(*NOTES TO SETUP VIRTUAL AXIS:
For the virtual axis setup, the encoders need their type changed from "simulation encoder" to "Encoder (Universal)".
In addition the scale factor needs to be changed to a numerator of 1 and denominator of fEncoderScaling which is 10,000 by default)
Care needs to be taken with scaling and setup of both real and virtual axes to ensure velocities are not too fast and axes have time to settle before they submit a "complete move"
Link the virtual encoder inputs to the Gap and Centre position calculations nGapSizePosition and nGapCentrePosition
Encoder needs to be set as ABSOLUTE
Encoder Mask has to be set to 0xFFFFFFFF otherwise UDINT will overflow
NOTES TO FB_SlitPair:
The instance of the function block should be called before the call of FB_Axis, so that it gets bExecute before FB_Axis
*)
FUNCTION_BLOCK FB_SlitPair
VAR_IN_OUT
    stBladeNegative: ST_AxisStruct; //Axis data of the negative blade
    stBladePositive: ST_AxisStruct; //Axis data of the positive blade
    stGapSize: ST_AxisStruct; //Axis data of the gap size
    stGapCentre: ST_AxisStruct; //Axis data of the gap centre
END_VAR
VAR_INPUT
    iGapSize: UINT; //Axis ID for the size of gap between slit blades
    iGapCentre: UINT; //Axis ID for the centre position of the gap formed by slit blades
    fEncoderScaling: LREAL := 10000.0; //default scaling denominator of 10000
    bAutoHome: BOOL := FALSE; //Blades homing is automatically done if they are not homed
    bAnticollisionEnable: BOOL := TRUE; //Blades anticollision option, only for when blades are moved independently
    fAnticollisionMargin: LREAL := 5.0; //Margin between the the blades for anticollision
END_VAR
VAR_OUTPUT
    bEnabled: BOOL := FALSE; //Enabled status of function
    bError: BOOL; //Error status of function
    bHoming: BOOL := FALSE; //TRUE if function is homing axes
END_VAR
VAR
    //Internal state machines
    eSlitPairState: E_SlitPairStates := E_SlitPairStates.eStartup; //Sequence steps for operating the slits
    eParameterCheck: E_AxisParamCheckState := E_AxisParamCheckState.eInit; //Sequence steps for checking params of virtual axes
    eSoftLimitsUpdate: E_SlitSoftLimits := E_SlitSoftLimits.eStart; //Sequence steps for update of soft limits for virtual axes

    //Internal statuses for logic
    bEnable: BOOL; //Enable/disable the slit set
    bReset: BOOL; //Reset the slit set
    bResetting: BOOL := FALSE; //TRUE if axis going through a reset
    bAxesEnabled: BOOL := FALSE; //TRUE if all axes enabled
    bBladesHomed: BOOL := FALSE; //TRUE if blade axes are calibrated
    bGapHomed: BOOL := FALSE; //TRUE if virtual axes are calibrated
    bBladesCoupled: BOOL := FALSE; //TRUE if both blade axes are coupled
    bBladesUncoupled: BOOL := FALSE; //TRUE if both blade axes are uncoupled
    bAxisErrorsPresent: BOOL := FALSE; //TRUE if error present on any real or virtual axis
    bUpdateSoftLimits: BOOL := FALSE; //TRUE if update of soft limits are being executed
    bHomingRequested: BOOL := FALSE; //TRUE if homing is requested for all axis
    bInvalidParamFound: BOOL := FALSE; //TRUE if startup finds atleast one invalid parameter
    fGapSizePosition: LREAL; //Virtual axis gap size calculated position
    nGapSizePosition AT %Q*: UDINT := 0; //Virtual axis gap size encoder position/counter
    fGapCentrePosition: LREAL; //Virtual axis gap centre calculated position
    nGapCentrePosition AT %Q*: UDINT := 0; //Virtual axis gap centre encoder position/counter
    nAutoErrorResetCounter: UINT := 0; //Error automatic reset counter
    iParamCheck: USINT := 1; //Index of current parameter to be validated
    rtrigSlitOperational: R_TRIG;
    rtrigVirtualAxisEnable: R_TRIG;
    rtrigVirtualAxisDisable: R_TRIG;
    rtrigVirtualAxisNotMoving: R_TRIG;
    fbResetCalibrationPositiveBlade: MC_Home;
    fbResetCalibrationNegativeBlade: MC_Home;
    fbResetCalibrationGapSize: MC_Home;
    fbResetCalibrationGapCentre: MC_Home;
END_VAR
VAR CONSTANT
    cSoftLimitDelta: LREAL := 0.05; //Delta between the softlimits of physical and virtual axes
    cMaxParams: USINT := 6;
    cParameters: ARRAY [1..cMaxParams] OF ST_AxisParamSpec := [ //Parameters required to be validated
        (eParam := E_AxisParameters.AxisEncoderScalingNumerator, fValue := 1.0),
        (eParam := E_AxisParameters.AxisEncoderScalingDenominator, fValue := 10000.0),
        (eParam := E_AxisParameters.AxisEncoderMask, fValue := 4294967295.0), //0xFFFFFFF = 4294967295.0
        (eParam := E_AxisParameters.AxisEncoderReferenceSystem, fValue := 1.0), //0.0 = INCREMENTAL, 1.0 = ABSOLUTE
        (eParam := E_AxisParameters.EnableLimitBackward, fValue := 1.0), //0.0 = FALSE, 1.0 = TRUE
        (eParam := E_AxisParameters.EnableLimitForward, fValue := 1.0)]; //0.0 = FALSE, 1.0 = TRUE
END_VAR

//Configure homing routine of virtual axes
stGapSize.stConfig.eHomeSeq := E_HomingRoutines.eHomeDirect;
stGapCentre.stConfig.eHomeSeq := E_HomingRoutines.eHomeDirect;

//Run actions for slit set
actErrorHandling(); //Error handling subroutine
actGapLimits(); //Set virtual axis limits to TRUE
actVirtualAxisPositions(); //Virtual axis encoder position subroutine
actUpdateStatus(); //Update statuses
actEnableAxes(); //Enable the axes
actClearCalibration(); //Clear calibration flag for all axes
mAnticollision(
    stBladeNegative := stBladeNegative,
    stBladePositive := stBladePositive); //Handle blades anticollision

CASE eSlitPairState OF
    E_SlitPairStates.eStartup:
        checkStartupParams(stGapSize, stGapCentre);
        IF eParameterCheck = E_AxisParamCheckState.eFinish THEN
            eSlitPairState := E_SlitPairStates.eInit;
        END_IF

    E_SlitPairStates.eInit:
        bEnabled := FALSE;
        IF bAxesEnabled AND bEnable THEN
            eSlitPairState := E_SlitPairStates.eInitClearGearing;
        END_IF

    E_SlitPairStates.eInitClearGearing:
        actClearSlitGearing();
        eSlitPairState := E_SlitPairStates.eInitGearOutCheck;

    E_SlitPairStates.eInitGearOutCheck: //Check gearout completion
        IF bBladesUncoupled THEN
            eSlitPairState := E_SlitPairStates.eCheckHomeStatus;
        END_IF

    E_SlitPairStates.eCheckHomeStatus: //If blades are already homed, skip to virtual homing, otherwise wait for manual/auto homing signal
        IF bBladesHomed THEN
            eSlitPairState := E_SlitPairStates.eHomeGap; //Skip to functioning
        ELSIF bAutoHome
            OR bHomingRequested
            OR (stGapSize.stControl.eCommand = E_MotionFunctions.eHome AND stGapSize.stControl.bExecute)
            OR (stGapCentre.stControl.eCommand = E_MotionFunctions.eHome AND stGapCentre.stControl.bExecute)
        THEN
            bHomingRequested := FALSE; //If homing fails do not automatically start homing again
            eSlitPairState := E_SlitPairStates.eHomeBlades;
        END_IF

    E_SlitPairStates.eHomeBlades: //Initiate homing of blade axes. Homing routine must be pre-configured by user
        stBladeNegative.stControl.eCommand := E_MotionFunctions.eHome;
        stBladePositive.stControl.eCommand := E_MotionFunctions.eHome;
        stBladeNegative.stControl.bExecute := TRUE;
        stBladePositive.stControl.bExecute := TRUE;
        bHoming := TRUE;
        eSlitPairState := E_SlitPairStates.eCheckBladeHomeComplete;

    E_SlitPairStates.eCheckBladeHomeComplete: //Wait for completion of blade homing routines or stop/halt command
        IF bBladesHomed AND NOT stBladeNegative.stStatus.bBusy AND NOT stBladePositive.stStatus.bBusy THEN
            eSlitPairState := E_SlitPairStates.eHomeGap;
            bHoming := FALSE;
        ELSIF stGapSize.stControl.bStop OR stGapCentre.stControl.bStop THEN
            stBladeNegative.stControl.bStop := TRUE;
            stBladePositive.stControl.bStop := TRUE;
            eSlitPairState := E_SlitPairStates.eCheckHomeStatus;
        ELSIF stGapSize.stControl.bHalt OR stGapCentre.stControl.bHalt THEN
            stBladeNegative.stControl.bHalt := TRUE;
            stBladePositive.stControl.bHalt := TRUE;
            eSlitPairState := E_SlitPairStates.eCheckHomeStatus;
        ELSIF (stBladeNegative.stStatus.nErrorID > 0) OR (stBladePositive.stStatus.nErrorID > 0) THEN
            eSlitPairState := E_SlitPairStates.eError;
        END_IF

    E_SlitPairStates.eHomeGap: //"Home" the virtual axes
        stGapSize.stConfig.eHomeSeq := E_HomingRoutines.eHomeDirect;
        stGapCentre.stConfig.eHomeSeq := E_HomingRoutines.eHomeDirect;
        stGapSize.stConfig.fHomePosition := fGapSizePosition;
        stGapCentre.stConfig.fHomePosition := fGapCentrePosition;
        stGapSize.stControl.eCommand := E_MotionFunctions.eHome;
        stGapCentre.stControl.eCommand := E_MotionFunctions.eHome;
        stGapSize.stControl.bExecute := TRUE;
        stGapCentre.stControl.bExecute := TRUE;
        eSlitPairState := E_SlitPairStates.eCheckGapHomeComplete;

    E_SlitPairStates.eCheckGapHomeComplete: //Wait for virtual homing completion
        IF bGapHomed AND NOT stGapSize.stStatus.bBusy AND NOT stGapCentre.stStatus.bBusy THEN
            eSlitPairState := E_SlitPairStates.eGearInSlits;
        END_IF

    E_SlitPairStates.eGearInSlits: //Setup gearing
        actSetupSlitGearing();
        eSlitPairState := E_SlitPairStates.eCheckGearInSlitsComplete;

    E_SlitPairStates.eCheckGearInSlitsComplete: //Wait for gearing complete
        IF bBladesCoupled THEN
            eSlitPairState := E_SlitPairStates.eSlitsOperational;
        ELSIF NOT stGapSize.stStatus.bEnabled AND NOT stGapCentre.stStatus.bEnabled THEN
            eSlitPairState := E_SlitPairStates.eErrorGearOut;
        END_IF

    E_SlitPairStates.eSlitsOperational: //SLITS OPERATIONAL - Monitor for any gear outs and re-gear when no busy blades
        bEnabled := TRUE;
        checkSoftLimits(stGapSize, stGapCentre); //Soft limits are updated when axes are stopped
        IF (NOT bBladesCoupled OR NOT bEnable) AND NOT stBladeNegative.stStatus.bBusy AND NOT stBladePositive.stStatus.bBusy THEN
            eSlitPairState := E_SlitPairStates.eGearOutBlades;
        END_IF
        IF (stGapSize.stControl.eCommand = E_MotionFunctions.eHome AND stGapSize.stControl.bExecute) OR
            (stGapCentre.stControl.eCommand = E_MotionFunctions.eHome AND stGapCentre.stControl.bExecute) THEN
            eSlitPairState := E_SlitPairStates.eGearOutBlades;
            bHomingRequested := TRUE;
        END_IF

    E_SlitPairStates.eGearOutBlades: //Clear any residual gearing
        actClearSlitGearing();
        eSlitPairState := E_SlitPairStates.eCheckGearOutComplete;

    E_SlitPairStates.eCheckGearOutComplete: //Check gearing cleared
        IF bBladesUncoupled THEN
            IF bHomingRequested THEN
                eSlitPairState := E_SlitPairStates.eResetCalibration;
                bEnabled := FALSE;
            ELSE
                eSlitPairState := E_SlitPairStates.eInit;
            END_IF
        END_IF

    E_SlitPairStates.eResetCalibration:
        IF checkResetCalibrationDone() THEN
            eSlitPairState := E_SlitPairStates.eCheckHomeStatus;
        ELSIF checkResetCalibrationFailed() THEN
            eSlitPairState := E_SlitPairStates.eError;
        END_IF

    E_SlitPairStates.eError: //ERROR STATE
        nAutoErrorResetCounter := 0;
        bError := TRUE;
        bEnabled := FALSE;
        IF bReset THEN
            bResetting := TRUE;
            eSlitPairState := E_SlitPairStates.eErrorGearOut;
        END_IF

    E_SlitPairStates.eErrorGearOut: //Try to clear issues
        actClearSlitGearing();
        eSlitPairState := E_SlitPairStates.eErrorGearOutCheck;

    E_SlitPairStates.eErrorGearOutCheck:
        IF bBladesUncoupled THEN
            eSlitPairState := E_SlitPairStates.eErrorResetAxes;
        END_IF

    E_SlitPairStates.eErrorResetAxes: //RESET ALL AXES
        stBladeNegative.stControl.bReset := TRUE;
        stBladePositive.stControl.bReset := TRUE;
        stGapSize.stControl.bReset := TRUE;
        stGapCentre.stControl.bReset := TRUE;
        nAutoErrorResetCounter := nAutoErrorResetCounter + 1;
        eSlitPairState := E_SlitPairStates.eErrorResetCheck;

    E_SlitPairStates.eErrorResetCheck:
        IF bAxisErrorsPresent THEN
            //If the errors persists after 10 auto reset, then manual intervention is required
            IF nAutoErrorResetCounter <= 10 THEN
                eSlitPairState := E_SlitPairStates.eErrorResetAxes;
            END_IF
        ELSE
            eSlitPairState := E_SlitPairStates.eInit;
            nAutoErrorResetCounter := 0;
            bError := FALSE;
            bResetting := FALSE;
        END_IF
END_CASE

bReset := FALSE;

ACTION actClearCalibration:
fbResetCalibrationPositiveBlade(
    Axis := stBladePositive.Axis,
    Execute := eSlitPairState = E_SlitPairStates.eResetCalibration,
    HomingMode := MC_HomingMode.MC_ResetCalibration);

fbResetCalibrationNegativeBlade(
    Axis := stBladeNegative.Axis,
    Execute := eSlitPairState = E_SlitPairStates.eResetCalibration,
    HomingMode := MC_HomingMode.MC_ResetCalibration);

fbResetCalibrationGapSize(
    Axis := stGapSize.Axis,
    Execute := eSlitPairState = E_SlitPairStates.eResetCalibration,
    HomingMode := MC_HomingMode.MC_ResetCalibration);

fbResetCalibrationGapCentre(
    Axis := stGapCentre.Axis,
    Execute := eSlitPairState = E_SlitPairStates.eResetCalibration,
    HomingMode := MC_HomingMode.MC_ResetCalibration);
END_ACTION

ACTION actClearSlitGearing:
//Action to send gearOut command to blade axes
stBladeNegative.stControl.eCommand := E_MotionFunctions.eGearOut;
stBladePositive.stControl.eCommand := E_MotionFunctions.eGearOut;
stBladeNegative.stControl.bExecute := TRUE;
stBladePositive.stControl.bExecute := TRUE;
END_ACTION

ACTION actEnableAxes:
//Enable all axes when one of the virtual axes is enabled
rtrigVirtualAxisEnable(CLK := stGapSize.stControl.bEnable OR stGapCentre.stControl.bEnable);

IF rtrigVirtualAxisEnable.Q THEN
    stBladePositive.stControl.bEnable := TRUE;
    stBladeNegative.stControl.bEnable := TRUE;
    stGapSize.stControl.bEnable := TRUE;
    stGapCentre.stControl.bEnable := TRUE;
    bEnable := TRUE;
END_IF

//Disable blade axes when both the virtuals are disabled
rtrigVirtualAxisDisable(CLK := NOT stGapSize.stControl.bEnable OR NOT stGapCentre.stControl.bEnable);

IF rtrigVirtualAxisDisable.Q THEN
    stBladePositive.stControl.bEnable := FALSE;
    stBladeNegative.stControl.bEnable := FALSE;
    stGapSize.stControl.bEnable := FALSE;
    stGapCentre.stControl.bEnable := FALSE;
END_IF

//Set Enable flag when all axes are enabled
bEnable := stBladePositive.stStatus.bEnabled AND stBladeNegative.stStatus.bEnabled
    AND stGapSize.stStatus.bEnabled AND stGapCentre.stStatus.bEnabled;
END_ACTION

ACTION actErrorHandling:
//Error handling for slit functionality
IF bResetting THEN //ignore setting in error state if FB going through a reset
    RETURN;
END_IF

//RESET - Use the reset from the virtual axes in order to reset the slits
bReset := stGapCentre.stControl.bReset OR stGapSize.stControl.bReset;

IF NOT bError AND bAxisErrorsPresent AND (stGapCentre.stStatus.bEnabled OR stGapSize.stStatus.bEnabled) THEN
    actStopAxes();
    eSlitPairState := E_SlitPairStates.eError;
END_IF

//Report error to virtual axes
IF eSlitPairState = E_SlitPairStates.eError THEN
    stGapCentre.stStatus.bError := TRUE;
    stGapSize.stStatus.bError := TRUE;
END_IF

IF bEnabled AND NOT bBladesHomed THEN
    eSlitPairState := E_SlitPairStates.eError;
END_IF
END_ACTION

ACTION actGapLimits:
//Set Virtual axes inputs to TRUE to enable movement
stGapSize.stInputs.bLimitBwd := stBladeNegative.stInputs.bLimitFwd OR stBladePositive.stInputs.bLimitBwd;
stGapSize.stInputs.bLimitFwd := stBladeNegative.stInputs.bLimitBwd OR stBladePositive.stInputs.bLimitFwd;
stGapCentre.stInputs.bLimitBwd := stBladeNegative.stInputs.bLimitFwd OR stBladePositive.stInputs.bLimitBwd;
stGapCentre.stInputs.bLimitFwd := stBladeNegative.stInputs.bLimitBwd OR stBladePositive.stInputs.bLimitFwd;
END_ACTION

ACTION actSetupSlitGearing:
//Setup multimaster gearing of negative blade
stBladeNegative.stControl.eCommand := E_MotionFunctions.eGearInMultiMaster;
stBladeNegative.stConfig.astMultiMasterAxis[1].nIndex := iGapSize;
stBladeNegative.stConfig.astMultiMasterAxis[1].fRatio := -0.5;
stBladeNegative.stConfig.astMultiMasterAxis[2].nIndex := iGapCentre;
stBladeNegative.stConfig.astMultiMasterAxis[2].fRatio := 1.0;
stBladeNegative.stConfig.astMultiMasterAxis[3].nIndex := iGapCentre;
stBladeNegative.stConfig.astMultiMasterAxis[3].fRatio := 0.0;
stBladeNegative.stConfig.astMultiMasterAxis[4].nIndex := iGapCentre;
stBladeNegative.stConfig.astMultiMasterAxis[4].fRatio := 0.0;
//Setup multimaster gearing of positive blade
stBladePositive.stControl.eCommand := E_MotionFunctions.eGearInMultiMaster;
stBladePositive.stConfig.astMultiMasterAxis[1].nIndex := iGapSize;
stBladePositive.stConfig.astMultiMasterAxis[1].fRatio := 0.5;
stBladePositive.stConfig.astMultiMasterAxis[2].nIndex := iGapCentre;
stBladePositive.stConfig.astMultiMasterAxis[2].fRatio := 1.0;
stBladePositive.stConfig.astMultiMasterAxis[3].nIndex := iGapCentre;
stBladePositive.stConfig.astMultiMasterAxis[3].fRatio := 0.0;
stBladePositive.stConfig.astMultiMasterAxis[4].nIndex := iGapCentre;
stBladePositive.stConfig.astMultiMasterAxis[4].fRatio := 0.0;
//Execute
stBladeNegative.stControl.bExecute := TRUE;
stBladePositive.stControl.bExecute := TRUE;
END_ACTION

ACTION actStopAxes:
//Stop all axes when in error (Abort movements)
stBladePositive.stControl.bStop := TRUE;
stBladeNegative.stControl.bStop := TRUE;
stGapSize.stControl.bStop := TRUE;
stGapCentre.stControl.bStop := TRUE;
END_ACTION

ACTION actUpdateSoftLimits:
//The soft limits of the virtual axes are updated everytime a movement has been accomplished.
//This is to avoid undesired errors if the user sets a target position which is not allowed

CASE eSoftLimitsUpdate OF

    E_SlitSoftLimits.eStart:
        eSoftLimitsUpdate := E_SlitSoftLimits.eWriteGapCentreFwd;

    E_SlitSoftLimits.eWriteGapCentreFwd:
        IF NOT stGapCentre.stStatus.bBusy AND NOT stGapSize.stStatus.bBusy THEN
            eSoftLimitsUpdate := E_SlitSoftLimits.eWriteGapCentreBwd;
            stGapCentre.stControl.bExecute := TRUE;
            stGapCentre.stControl.eCommand := E_MotionFunctions.eWriteParameter;
            stGapCentre.stConfig.eAxisParameters := E_AxisParameters.SWLimitForward;
            stGapCentre.stConfig.fWriteAxisParameter := stBladePositive.stConfig.fMaxSoftPosLimit
                - ABS(stGapCentre.stStatus.fActPosition - stBladePositive.stStatus.fActPosition)
                - cSoftLimitDelta;
        END_IF

    E_SlitSoftLimits.eWriteGapCentreBwd:
        IF stGapCentre.stStatus.bDone AND NOT stGapCentre.stControl.bExecute THEN
            eSoftLimitsUpdate := E_SlitSoftLimits.eWriteGapSizeFwd;
            stGapCentre.stControl.bExecute := TRUE;
            stGapCentre.stControl.eCommand := E_MotionFunctions.eWriteParameter;
            stGapCentre.stConfig.eAxisParameters := E_AxisParameters.SWLimitBackward;
            stGapCentre.stConfig.fWriteAxisParameter := stBladeNegative.stConfig.fMinSoftPosLimit
                + ABS(stGapCentre.stStatus.fActPosition - stBladeNegative.stStatus.fActPosition)
                + cSoftLimitDelta;
        END_IF

    E_SlitSoftLimits.eWriteGapSizeFwd:
        IF stGapCentre.stStatus.bDone AND NOT stGapCentre.stControl.bExecute THEN
            eSoftLimitsUpdate := E_SlitSoftLimits.eFinish;
            stGapSize.stControl.bExecute := TRUE;
            stGapSize.stControl.eCommand := E_MotionFunctions.eWriteParameter;
            stGapSize.stConfig.eAxisParameters := E_AxisParameters.SWLimitForward;
            stGapSize.stConfig.fWriteAxisParameter := 2.0 * MAX(MIN(
                ABS(stBladePositive.stConfig.fMaxSoftPosLimit - stGapCentre.stStatus.fActPosition),
                ABS(stBladeNegative.stConfig.fMinSoftPosLimit - stGapCentre.stStatus.fActPosition))
                - cSoftLimitDelta,
                0.0);
        END_IF

    E_SlitSoftLimits.eFinish:
        IF stGapSize.stStatus.bDone AND NOT stGapSize.stControl.bExecute THEN
            eSoftLimitsUpdate := E_SlitSoftLimits.eStart;
            bUpdateSoftLimits := FALSE;
        END_IF

END_CASE
END_ACTION

ACTION actUpdateStatus:
bAxesEnabled := checkAllAxesEnabled(stBladeNegative, stBladePositive, stGapSize, stGapCentre);
bBladesHomed := checkBladesHomed(stBladeNegative, stBladePositive);
bGapHomed := checkGapHomed(stGapSize, stGapCentre);
bBladesCoupled := checkBladesCoupled(stBladeNegative, stBladePositive);
bBladesUncoupled := checkBladesUncoupled(stBladeNegative, stBladePositive);
bAxisErrorsPresent := checkAnyAxisHasError(stBladeNegative, stBladePositive, stGapSize, stGapCentre);
END_ACTION

ACTION actVirtualAxisPositions:
(*Calculate virtual axes positions and convert to UDINT.
Conversion to UDINT is prohibited if it would exceed UDINT max value of 4,294,967,295.
If this is not done, it can cause overflow when connected to the encoder input and hard-crash the PLC which will only recover with a power cycle.
To preserve decimal position data of the LREAL (i.e. anything <1mm) it is necessary to scale the value before converting to UDINT.
This can be reversed with the correct scaling at the NC encoder level.
*)
fGapSizePosition := stBladePositive.stStatus.fActPosition - stBladeNegative.stStatus.fActPosition;
fGapCentrePosition := (stBladePositive.stStatus.fActPosition + stBladeNegative.stStatus.fActPosition) / 2;

IF bBladesHomed THEN
    IF ABS(fGapSizePosition) < 100000 THEN
        nGapSizePosition := LREAL_TO_UDINT(fGapSizePosition*fEncoderScaling);
    END_IF
    IF ABS(fGapCentrePosition) < 100000 THEN
        nGapCentrePosition := LREAL_TO_UDINT(fGapCentrePosition*fEncoderScaling);
    END_IF
END_IF
END_ACTION

(*Method to check if all axes (real and virtual) are enabled.
Only returns TRUE if BOTH blades are homed*)
METHOD PRIVATE checkAllAxesEnabled: BOOL
VAR_IN_OUT
    stBladeNegative: ST_AxisStruct; //Axis data of the negative blade
    stBladePositive: ST_AxisStruct; //Axis data of the positive blade
    stGapSize: ST_AxisStruct; //Axis data of the gap size
    stGapCentre: ST_AxisStruct; //Axis data of the gap centre
END_VAR
checkAllAxesEnabled := stBladeNegative.stStatus.bEnabled
    AND stBladePositive.stStatus.bEnabled
    AND stGapSize.stStatus.bEnabled
    AND stGapCentre.stStatus.bEnabled;
END_METHOD

(*Method to check if an error is present on any axis.
Returns TRUE if an error is present on any axis *)
METHOD PRIVATE checkAnyAxisHasError: BOOL
VAR_IN_OUT
    stBladeNegative: ST_AxisStruct; //Axis data of the negative blade
    stBladePositive: ST_AxisStruct; //Axis data of the positive blade
    stGapSize: ST_AxisStruct; //Axis data of the gap size
    stGapCentre: ST_AxisStruct; //Axis data of the gap centre
END_VAR
checkAnyAxisHasError := stGapSize.stStatus.bError
    OR stGapCentre.stStatus.bError
    OR stBladeNegative.stStatus.bError
    OR stBladePositive.stStatus.bError;
END_METHOD

(*Method to check if both blades are coupled to the virtual axes.
Only returns TRUE if BOTH blades are coupled *)
METHOD PRIVATE checkBladesCoupled: BOOL
VAR_IN_OUT
    stBladeNegative: ST_AxisStruct; //Axis data of the negative blade
    stBladePositive: ST_AxisStruct; //Axis data of the positive blade
END_VAR
checkBladesCoupled := stBladeNegative.stStatus.bGeared AND stBladePositive.stStatus.bGeared;
END_METHOD

(*Method to check if blade axes are homed/have the calibration flag.
Only returns TRUE if BOTH blades are homed*)
METHOD PRIVATE checkBladesHomed: BOOL
VAR_IN_OUT
    stBladeNegative: ST_AxisStruct; //Axis data of the negative blade
    stBladePositive: ST_AxisStruct; //Axis data of the positive blade
END_VAR
checkBladesHomed := stBladeNegative.stStatus.bHomed AND stBladePositive.stStatus.bHomed;
END_METHOD

(*Method to check if both blades are uncoupled from the virtual axes.
Only returns TRUE if BOTH blades are uncoupled *)
METHOD PRIVATE checkBladesUncoupled: BOOL
VAR_IN_OUT
    stBladeNegative: ST_AxisStruct; //Axis data of the negative blade
    stBladePositive: ST_AxisStruct; //Axis data of the positive blade
END_VAR
checkBladesUncoupled := NOT (stBladeNegative.stStatus.bGeared OR stBladePositive.stStatus.bGeared);
END_METHOD

(*Method to check if the virtual axes for gap size and gap centre are homed/the calibration flag is present.
Only returns TRUE if BOTH virtual axes are homed *)
METHOD PRIVATE checkGapHomed: BOOL
VAR_IN_OUT
    stGapSize: ST_AxisStruct; //Axis data of the gap size
    stGapCentre: ST_AxisStruct; //Axis data of the gap size
END_VAR
checkGapHomed := stGapSize.stStatus.bHomed AND stGapCentre.stStatus.bHomed;
END_METHOD

METHOD PRIVATE checkResetCalibrationDone : BOOL
VAR_INPUT
END_VAR
checkResetCalibrationDone := NOT fbResetCalibrationPositiveBlade.Busy
    AND NOT fbResetCalibrationNegativeBlade.Busy
    AND NOT fbResetCalibrationGapSize.Busy
    AND NOT fbResetCalibrationGapCentre.Busy
    AND NOT bBladesHomed
    AND NOT bGapHomed;
END_METHOD

METHOD PRIVATE checkResetCalibrationFailed : BOOL
VAR_INPUT
END_VAR
checkResetCalibrationFailed := fbResetCalibrationPositiveBlade.Error
    OR fbResetCalibrationNegativeBlade.Error
    OR fbResetCalibrationGapSize.Error
    OR fbResetCalibrationGapCentre.Error
    OR fbResetCalibrationPositiveBlade.CommandAborted
    OR fbResetCalibrationNegativeBlade.CommandAborted
    OR fbResetCalibrationGapSize.CommandAborted
    OR fbResetCalibrationGapCentre.CommandAborted;
END_METHOD

METHOD PRIVATE checkSoftLimits
VAR_IN_OUT
    stGapSize: ST_AxisStruct; //Axis data of the gap size
    stGapCentre: ST_AxisStruct; //Axis data of the gap centre
END_VAR
rtrigVirtualAxisNotMoving(CLK := NOT stGapCentre.stStatus.bMoving AND NOT stGapSize.stStatus.bMoving);
rtrigSlitOperational(CLK := eSlitPairState = E_SlitPairStates.eSlitsOperational);

IF rtrigVirtualAxisNotMoving.Q OR rtrigSlitOperational.Q THEN
    bUpdateSoftLimits := TRUE;
END_IF

IF bUpdateSoftLimits THEN
    actUpdateSoftLimits();
END_IF
END_METHOD

METHOD PRIVATE checkStartupParams
VAR_IN_OUT
    stGapSize: ST_AxisStruct; //Axis data of the gap size
    stGapCentre: ST_AxisStruct; //Axis data of the gap centre
END_VAR
VAR
    sWarnMsg: T_MaxString;
END_VAR
CASE eParameterCheck OF
    E_AxisParamCheckState.eInit:
        //Wait for axis initialization
        IF NOT (stGapSize.stStatus.bAxisInitialized AND stGapCentre.stStatus.bAxisInitialized) THEN
            RETURN;
        END_IF

        iParamCheck := 1;
        eParameterCheck := E_AxisParamCheckState.eSelectParam;

    E_AxisParamCheckState.eSelectParam:
        stGapSize.stConfig.eAxisParameters := cParameters[iParamCheck].eParam;
        stGapSize.stControl.eCommand := E_MotionFunctions.eReadParameter;
        stGapSize.stControl.bExecute := TRUE;

        stGapCentre.stConfig.eAxisParameters := cParameters[iParamCheck].eParam;
        stGapCentre.stControl.eCommand := E_MotionFunctions.eReadParameter;
        stGapCentre.stControl.bExecute := TRUE;

        eParameterCheck := E_AxisParamCheckState.eWaitRead;

    E_AxisParamCheckState.eWaitRead:
        //Parameter reading still in progress
        IF stGapSize.stStatus.bBusy OR stGapCentre.stStatus.bBusy THEN
            RETURN;
        END_IF

        eParameterCheck := E_AxisParamCheckState.eCheck;

    E_AxisParamCheckState.eCheck:
        IF stGapSize.stConfig.fReadAxisParameter = cParameters[iParamCheck].fValue
            AND stGapCentre.stConfig.fReadAxisParameter = cParameters[iParamCheck].fValue
        THEN
            eParameterCheck := E_AxisParamCheckState.eParamValid;
        ELSE
            eParameterCheck := E_AxisParamCheckState.eParamInvalid;
        END_IF

    E_AxisParamCheckState.eParamValid:
        eParameterCheck := E_AxisParamCheckState.eNext;

    E_AxisParamCheckState.eParamInvalid:
        //Gap Size
        IF stGapSize.stConfig.fReadAxisParameter <> cParameters[iParamCheck].fValue THEN
            sWarnMsg := CONCAT(
                STR1 := 'Slit virtual axis Gap Size (AxisId=%d) has an invalid parameter of ',
                STR2 := TO_STRING(cParameters[iParamCheck].eParam));

            ADSLOGDINT(
                msgCtrlMask := ADSLOG_MSGTYPE_WARN,
                msgFmtStr := sWarnMsg,
                dintArg := TO_DINT(iGapSize));
        END_IF
        //Gap Centre
        IF stGapCentre.stConfig.fReadAxisParameter <> cParameters[iParamCheck].fValue THEN
            sWarnMsg := CONCAT(
                STR1 := 'Slit virtual axis Gap Centre (AxisId=%d) has an invalid parameter of ',
                STR2 := TO_STRING(cParameters[iParamCheck].eParam));

            ADSLOGDINT(
                msgCtrlMask := ADSLOG_MSGTYPE_WARN,
                msgFmtStr := sWarnMsg,
                dintArg := TO_DINT(iGapCentre));
        END_IF
        bInvalidParamFound := TRUE;

        eParameterCheck := E_AxisParamCheckState.eNext;

    E_AxisParamCheckState.eNext:
        IF iParamCheck = cMaxParams THEN
            IF NOT bInvalidParamFound THEN
                ADSLOGSTR(
                    msgCtrlMask := ADSLOG_MSGTYPE_LOG,
                    msgFmtStr := 'Slit all parameters of both virtual axes are valid',
                    strArg := '');
            END_IF
            eParameterCheck := E_AxisParamCheckState.eFinish;
        ELSE
            ;
            iParamCheck := iParamCheck + 1;
            eParameterCheck := E_AxisParamCheckState.eSelectParam;
        END_IF


    E_AxisParamCheckState.eFinish:
        ;

END_CASE
END_METHOD

METHOD PRIVATE mAntiCollision
VAR_IN_OUT
    stBladeNegative: ST_AxisStruct; //Axis data of the negative blade
    stBladePositive: ST_AxisStruct; //Axis data of the positive blade
END_VAR
VAR
    fNegativeBladePosWithMargin: LREAL;
    fPositiveBladePosWithMargin: LREAL;
END_VAR
//Return early if preconditions are not met
IF NOT (bBladesHomed
    AND bBladesUncoupled
    AND bAnticollisionEnable)
THEN
    RETURN;
END_IF

//Negative Blade

fPositiveBladePosWithMargin := (stBladePositive.stStatus.fActPosition - fAnticollisionMargin);

//If executing absolute / relative movement commands also check target position
IF stBladeNegative.stControl.bExecute THEN
    CASE stBladeNegative.stControl.eCommand OF

        E_MotionFunctions.eMoveAbsolute:
            stBladeNegative.stControl.bInterlockFwd S= stBladeNegative.stControl.fPosition
                >= fPositiveBladePosWithMargin;

        E_MotionFunctions.eMoveRelative:
            stBladeNegative.stControl.bInterlockFwd S= (stBladeNegative.stControl.fPosition
                + stBladeNegative.stStatus.fActPosition)
                >= fPositiveBladePosWithMargin;

    END_CASE
END_IF

//Check if current position is outside the anticollision margin
stBladeNegative.stControl.bInterlockFwd S= stBladeNegative.stStatus.fActPosition
    >= fPositiveBladePosWithMargin;

//Positive Blade

fNegativeBladePosWithMargin := (stBladeNegative.stStatus.fActPosition + fAnticollisionMargin);

//If executing absolute / relative movement commands also check target position
IF stBladePositive.stControl.bExecute THEN
    CASE stBladePositive.stControl.eCommand OF

        E_MotionFunctions.eMoveAbsolute:
            stBladePositive.stControl.bInterlockBwd S= stBladePositive.stControl.fPosition
                <= fNegativeBladePosWithMargin;

        E_MotionFunctions.eMoveRelative:
            stBladePositive.stControl.bInterlockBwd S= (stBladePositive.stControl.fPosition
                + stBladePositive.stStatus.fActPosition)
                <= fNegativeBladePosWithMargin;

    END_CASE
END_IF

//Check if current position is outside the anticollision margin
stBladePositive.stControl.bInterlockBwd S= stBladePositive.stStatus.fActPosition
    <= fNegativeBladePosWithMargin;
END_METHOD

END_FUNCTION_BLOCK

(* stored: Version 1.1.0.1
   POU FB_SlitPair: Id {e905bacc-19e9-06c3-04ae-f4fd4f34065e}, SpecialFunc None
   Action actClearCalibration: Id {ebc4e684-09cb-0ff6-2420-a784d5e2b2e0}
   Action actClearSlitGearing: Id {1b3caf4f-ddef-035c-06c2-b31f09d8bc8e}
   Action actEnableAxes: Id {1879c38a-aecf-0e8c-2a58-959e274ebc63}
   Action actErrorHandling: Id {d6af18ad-d698-0d90-0e47-da58345e8c10}
   Action actGapLimits: Id {def3d604-4e23-0583-39ed-61c5876cfc85}
   Action actSetupSlitGearing: Id {7713a838-7a24-0b22-0e20-e71c745ddc61}
   Action actStopAxes: Id {83b4f1fe-f696-016b-03db-3bcff9089f7d}
   Action actUpdateSoftLimits: Id {35e948c5-fa3a-0897-288a-c8995c0599d0}
   Action actUpdateStatus: Id {41ae3d05-bdbb-08b3-3ad3-022e54908169}
   Action actVirtualAxisPositions: Id {7f6698b5-ef89-01d2-091a-1167e8f62f6e}
   Method checkAllAxesEnabled: Id {68815ab2-933a-0cf6-0de8-cc7494d09118}
   Method checkAnyAxisHasError: Id {38d2d046-b549-0765-1487-87302195ffc6}
   Method checkBladesCoupled: Id {4d5a8473-6708-0035-3843-638ffe259036}
   Method checkBladesHomed: Id {81c53f0d-71e1-0f29-1da7-da19807b67a4}
   Method checkBladesUncoupled: Id {c279ba5c-ed4a-0e71-2fa2-767db0f1b8c8}
   Method checkGapHomed: Id {4449923d-b61f-063b-337f-e765d5643490}
   Method checkResetCalibrationDone: Id {c8bd46bd-3fc2-0717-0d3e-69d1ca8c8ae0}
   Method checkResetCalibrationFailed: Id {aacfc6b7-b4c3-0651-27cc-e962cf487e92}
   Method checkSoftLimits: Id {7b17dbf3-e1d6-0a6e-1aa4-6cded47f1f4b}
   Method checkStartupParams: Id {0a75b0a0-5874-0b4b-15f1-5347be377ef8}
   Method mAntiCollision: Id {ceddaf27-2734-0a8a-1c66-3bf942e8b7e9} *)
